VISUALIZATION HMI_Test  // 1024x768
END_VISUALIZATION

(* stored: Version 1.1.0.1
   Visu HMI_Test: Id {fdee1b17-8c6d-460a-8710-38e7d6dd4862} *)
